(* Logix 5000 project; controller ProyectoIntegrador Emulate 5570 rev 30.11; software revision 30.00 *)

TASK MainTask (continuous, watchdog 500 ms) : MainProgram

MODULES
   Local : Emulate 5570 (ICP 2, rev 30.11)
      IO_module : vendor 1 type 0 code 15 (ICP 3, rev 1.1, Output RPI 150 ms)
END_MODULES

PROGRAM MainProgram   (* main routine MainRoutine *)
VAR
   Step_000 : SFC_STEP := (Status := 16#0020_0000, PauseTimer := 1);
   Step_002 : SFC_STEP := (Status := 16#0020_0000, PauseTimer := 1);
   Step_004 : SFC_STEP := (Status := 16#0020_0000, PauseTimer := 1);
   Step_005 : SFC_STEP := (Status := 16#0020_0000, PauseTimer := 1);
   Step_006 : SFC_STEP := (Status := 16#0020_0000, PauseTimer := 1);
   Step_007 : SFC_STEP := (Status := 16#0020_0000, PauseTimer := 1);
   Step_008 : SFC_STEP := (Status := 16#0020_0000, PauseTimer := 1);
   Step_009 : SFC_STEP := (Status := 16#0020_0000, PauseTimer := 1);
   Tran_001 : BOOL;
   Tran_002 : BOOL;
   Tran_003 : BOOL;
   Tran_004 : BOOL;
   Tran_005 : BOOL;
   Tran_006 : BOOL;
END_VAR

ROUTINE Main   (* sequential function chart *)
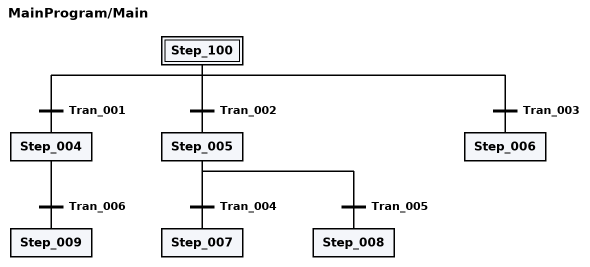
   INITIAL_STEP Step_100:
   END_STEP
   TRANSITION Tran_001 FROM Step_100 TO Step_004
      := 
   END_TRANSITION
   TRANSITION Tran_002 FROM Step_100 TO Step_005
      := 
   END_TRANSITION
   TRANSITION Tran_003 FROM Step_100 TO Step_006
      := 
   END_TRANSITION
   STEP Step_004:
   END_STEP
   STEP Step_005:
   END_STEP
   TRANSITION Tran_006 FROM Step_004 TO Step_009
      := 
   END_TRANSITION
   STEP Step_006:
   END_STEP
   STEP Step_009:
   END_STEP
   TRANSITION Tran_004 FROM Step_005 TO Step_007
      := 
   END_TRANSITION
   TRANSITION Tran_005 FROM Step_005 TO Step_008
      := 
   END_TRANSITION
   STEP Step_007:
   END_STEP
   STEP Step_008:
   END_STEP
END_ROUTINE

ROUTINE MainRoutine   (* ladder *)
END_ROUTINE

ROUTINE T001   (* structured text *)
   S_class = isGreen
END_ROUTINE
END_PROGRAM
